// TwinCAT 3 PLC project DomainTemplate
// ProgramVersion: 3.1.4026.9
// libraries:
//   Tc2_Standard, * (Beckhoff Automation GmbH)
//   Tc2_System, * (Beckhoff Automation GmbH)
//   Broadcast, * (_)
//   Debug, * (_)
//   Domains, * (_)
//   Flags, * (_)
//   Parameters, * (_)
//   Results, * (_)
//   Rt, * (_)
//   States, * (_)
//   Strings, * (_)
//   Tags, * (_)
//   Utils, * (_)
// project tree:
//   Domain%28Copy and rename%29/Ctx/ ExampleDomain_Hmi.TcDUT (not stored), ExampleDomain_Io.TcDUT (not stored), ExampleDomain_Priv.TcDUT (not stored), ExampleDomain_States.TcPOU (not stored)
//   Domain%28Copy and rename%29/Ctx/Io/ ExampleDomain_Io_In.TcDUT (not stored), ExampleDomain_Io_Out.TcDUT (not stored)
//   Domain%28Copy and rename%29/ ExampleDomain.TcPOU (not stored), ExampleDomain_Ctx.TcDUT (not stored)
//   Domain%28Copy and rename%29/State/ ExampleDomain_ExampleState.TcPOU (not stored), _ExampleDomain_State.TcPOU (not stored)
//   Domain%28Copy and rename%29/Ui/ ExampleDomain_StatusText.TcPOU (not stored)
//   / README.TcPOU
// (motion and I/O tree: see PLC project broadcast)
// real-time tasks:
//   TASK PlcTask: cycle T#10ms, priority 20, ADS port 350
//   TASK VISU_TASK: cycle T#200000us, priority 30, ADS port 351

// ---- README.TcPOU
PROGRAM README

(*
This is a template for a Domain object. Copy this folder to your project and rename its files to suit your application.
The 'ExampleDomain' domain is just a placeholder. You folder should be named e.g. 'ConveyorMgr' and then it should have the following structure:

ConveyorMgr
|
|-- Ctx
|   |-- Io
|   |   |-- ConveyorMgr_Io_In (STRUCT)
|   |   |-- ConveyorMgr_Io_Out (STRUCT)
|   |
|   |-- ConveyorMgr_Hmi (STRUCT)
|   |-- ConveyorMgr_Io (STRUCT)
|   |-- ConveyorMgr_Priv (STRUCT)
|   |-- ConveyorMgr_States (FB)
|
|-- State
|   |-- _ConveyorMgr_State (FB)
|   |-- ConveyorMgr_ExampleState (FB)
|
|-- Ui
|   |-- Visu
|   |
|   |-- ConveyorManager_StatusText (FB)
|
|-- ConveyorMgr (FB)
|-- ConveyorMgr_Ctx (STRUCT)

*)

END_PROGRAM
